// TIA Portal V20 export
FUNCTION "FC_1" : Void   // FC1, LAD
{ S7_Optimized_Access := 'TRUE' }
// stored: SetENOAutomatically false
BEGIN

REGION Network 1
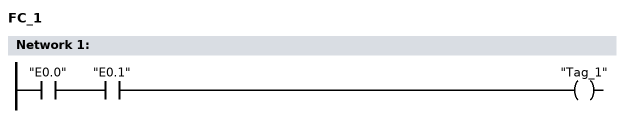
   RUNG wire#powerrail
      Contact( "E0.0" )
      Contact( "E0.1" )
      Coil( "Tag_1" )
   END_RUNG
   // the same network as SCL:
   "Tag_1" := "E0.0" AND "E0.1";
END_REGION
END_FUNCTION
